// TIA Portal project "LabSupervision" (V16)

(* hardware
DEVICE "S71500/ET200MP station_1"  S7-1500 station
   slot 0: "Perfil soporte_0"  Rack  6ES7 590-1***0-0AA0
   slot 0: "PM 70W 120/230VAC"  PM 70W 120/230VAC  6EP1332-4BA00
   slot 1: "PLC_1"  CPU 1511-1 PN  6ES7 511-1AK00-0AB0  V1.0
      slot 3: "Display de la CPU_1"  6ES7591-1XA00-0AA0
      slot 32768: "Interfaz PROFINET_1"  X1
   slot 2: "CM 1542-5_1"  CM 1542-5  6GK7 542-5DX00-0XE0  V1.0
   slot 3: "DI 16x24VDC HF_1"  DI 16x24VDC HF  6ES7 521-1BH00-0AB0  V1.0
   slot 4: "DQ 16x24VDC/0.5A HF_1"  DQ 16x24VDC/0.5A HF  6ES7 522-1BH01-0AB0  V1.0
   slot 5: "AI 8xU/I/RTD/TC ST_1"  AI 8xU/I/RTD/TC ST  6ES7 531-7KF00-0AB0  V1.0
   slot 6: "AQ 4xU/I ST_1"  AQ 4xU/I ST  6ES7 532-5HD00-0AB0  V1.0
DEVICE "HMI_1"  KTP600 Basic color PN
   slot 0: "HMI_1"  KTP600 Basic color PN  6AV6 647-0AD11-3AX0  12.0.0.0
   slot 1: "HMI_RT_1"  KTP600 Basic color PN  6AV6 647-0AD11-3AX0  12.0.0.0
   slot 5: "HMI_1.IE_CP_1"  PROFINET Interface  12.0.0.0
      slot 1: "Interfaz PROFINET_1"  PROFINET Interface
         slot 1: "Port_1"  Port
DEVICE "PC-System_1"  SIMATIC PC station
   slot 0: "Estación PC SIMATIC"  Rail  SIMATIC PC-Station  V1.0
      slot 125: "Stationmanager"  Station_Manager  V6.0.4
   slot 1: "HMI_RT_2"  WinCC RT Professional  6AV2 105-0xxxx-xxxx  16.0.0.0
   slot 2: "IE general_1"  IE General  IE_CP  V8.2.0
DEVICE "SINAMICS G_1"  Sinamics.Device
   slot 0: "	_0"  Rail  SinamicsG120RackPN
   slot 0: "Accionamiento_1"  G120 CU240E-2 PN  6SL3244-0BB12-1FA0  4.7.6
      slot 1: "Interfaz PROFINET"  MDD-SinamicsG120-P
   slot 3: "PM240-2 IP20"  PM240-2 IP20  6SL3210-1PB13-8ULx  -
*)

// ===== PLC "PLC_1"  CPU 1511-1 PN =====

VAR_GLOBAL   // PLC tag table "Tabla de variables estándar"
   "Señal_Intermitente" AT %Q0.0 : Bool;
   "STAR" AT %M0.0 : Bool;
   "Potenciometro" AT %MW2 : Int;
   "Nivel_Actual" AT %QW2 : Int;
   "pot_Normalizado" AT %MD2 : Real;
   "Alarma_Nivel_Alto" AT %Q0.1 : Bool;
   "Alarma_Nivel_Bajo" AT %Q0.2 : Bool;
   "Stop" AT %I0.1 : Bool;
   "Paro_Emergencia" AT %I0.3 : Bool;
   "BomBa" AT %Q0.3 : Bool;
   "Sensor_Nivel_Alto" AT %I0.4 : Bool;
   "Sensor_Nivel_Bajo" AT %I0.5 : Bool;
   "Sistema" AT %M0.7 : Bool;
   "Bomba_Agua" AT %M0.2 : Bool;
   "Referencia" AT %MW6 : Int;
   "Nivel_Alcanzado" AT %Q0.6 : Bool;
   "Delante" AT %M0.6 : Bool;
   "Atras" AT %M1.0 : Bool;
   "RPM" AT %M8.0 : LReal;
END_VAR

DATA_BLOCK "Bloque_1_DB"   // DB5
{ S7_Optimized_Access := 'TRUE' }
VERSION : 0.1
// stored: InstanceOfName Bloque_1
"Bloque_1"
BEGIN
END_DATA_BLOCK

DATA_BLOCK "Base_Datos"   // DB8
{ S7_Optimized_Access := 'TRUE' }
VERSION : 0.1
   VAR
      RPM : Real;
      NivelLeidoInt : Real;
      Revoluciones_datos : Real;
   END_VAR
BEGIN
END_DATA_BLOCK

// folder: System blocks/Program resources

DATA_BLOCK "Encender"   // DB1
{ S7_Optimized_Access := 'TRUE' }
AUTHOR : Simatic
FAMILY : IEC
NAME : IEC_TMR
VERSION : 1.0
// stored: InstanceOfName IEC_TIMER
"IEC_TIMER"
BEGIN
END_DATA_BLOCK

DATA_BLOCK "apagar"   // DB2
{ S7_Optimized_Access := 'TRUE' }
AUTHOR : Simatic
FAMILY : IEC
NAME : IEC_TMR
VERSION : 1.0
// stored: InstanceOfName IEC_TIMER
"IEC_TIMER"
BEGIN
END_DATA_BLOCK

DATA_BLOCK "IEC_Timer_0_DB"   // DB3
{ S7_Optimized_Access := 'TRUE' }
AUTHOR : Simatic
FAMILY : IEC
NAME : IEC_TMR
VERSION : 1.0
// stored: InstanceOfName IEC_TIMER
"IEC_TIMER"
BEGIN
END_DATA_BLOCK

DATA_BLOCK "IEC_Timer_0_DB_1"   // DB6
{ S7_Optimized_Access := 'TRUE' }
AUTHOR : Simatic
FAMILY : IEC
NAME : IEC_TMR
VERSION : 1.0
// stored: InstanceOfName IEC_TIMER
"IEC_TIMER"
BEGIN
END_DATA_BLOCK

DATA_BLOCK "IEC_Timer_0_DB_2"   // DB7
{ S7_Optimized_Access := 'TRUE' }
AUTHOR : Simatic
FAMILY : IEC
NAME : IEC_TMR
VERSION : 1.0
// stored: InstanceOfName IEC_TIMER
"IEC_TIMER"
BEGIN
END_DATA_BLOCK

// folder: (top level)

DATA_BLOCK "TO_SpeedAxis_1"   // DB4, Motion_DB
{ S7_Optimized_Access := 'TRUE' }
AUTHOR : SIMATIC
FAMILY : MC_1500
VERSION : 1.0
// stored: InstanceOfName TO_SpeedAxis
"TO_SpeedAxis"
BEGIN
   DynamicLimits.MaxAcceleration := 1000.0;
   DynamicLimits.MaxDeceleration := 1000.0;
   DynamicLimits.MaxJerk := 20000.0;
   DynamicDefaults.Acceleration := 200.0;
   DynamicDefaults.Deceleration := 200.0;
   DynamicDefaults.Jerk := 4000.0;
   DynamicDefaults.EmergencyDeceleration := 1000.0;
   Actor.Interface.AddressOut := 256;
   Actor.Interface.AddressIn := 256;
END_DATA_BLOCK

FUNCTION_BLOCK "Bloque_1"   // FB1, LAD
{ S7_Optimized_Access := 'TRUE' }
VERSION : 0.1
   VAR
      MC_POWER_Instance : MC_POWER;
      MC_RESET_Instance : MC_RESET;
      MC_MOVEJOG_Instance : MC_MOVEJOG;
   END_VAR
BEGIN

REGION Network 1
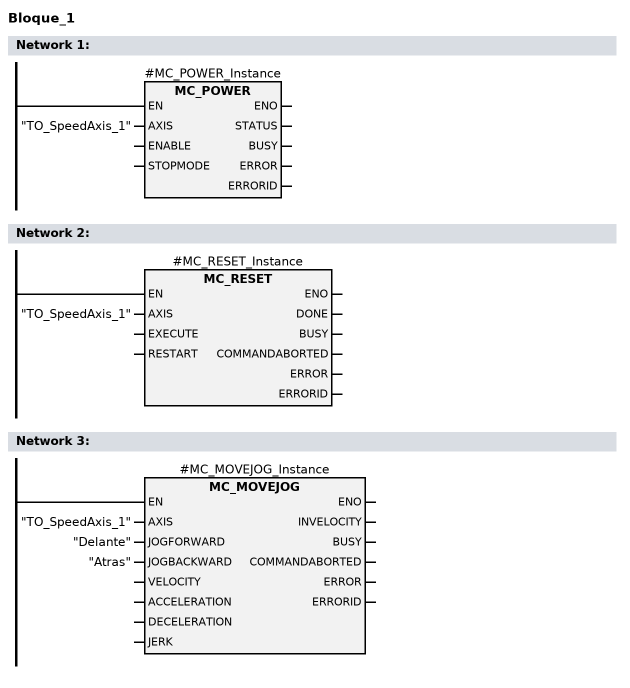
   #MC_POWER_Instance(Axis := "TO_SpeedAxis_1");   // MC_POWER
END_REGION

REGION Network 2
   #MC_RESET_Instance(Axis := "TO_SpeedAxis_1");   // MC_RESET
END_REGION

REGION Network 3
   #MC_MOVEJOG_Instance(Axis := "TO_SpeedAxis_1", JogForward := "Delante", JogBackward := "Atras");   // MC_MOVEJOG
END_REGION
END_FUNCTION_BLOCK

ORGANIZATION_BLOCK "Main"   // OB1, LAD, ProgramCycle
TITLE = "Main Program Sweep (Cycle)"
{ S7_Optimized_Access := 'TRUE' }
VERSION : 0.1
   VAR_INPUT
      Initial_Call : Bool;   // Initial call of this OB
      Remanence : Bool;   // =True, if remanent data are available
   END_VAR
   VAR_TEMP
      Temp_1 : Bool;
      Activar_Bomba : Bool;
      intermitencia : Bool;
   END_VAR
   VAR_TEMP   // added for the SCL form of the ladder/FBD networks
      _w1 : Bool;
   END_VAR
BEGIN

REGION Network 1: Normalizar Señal
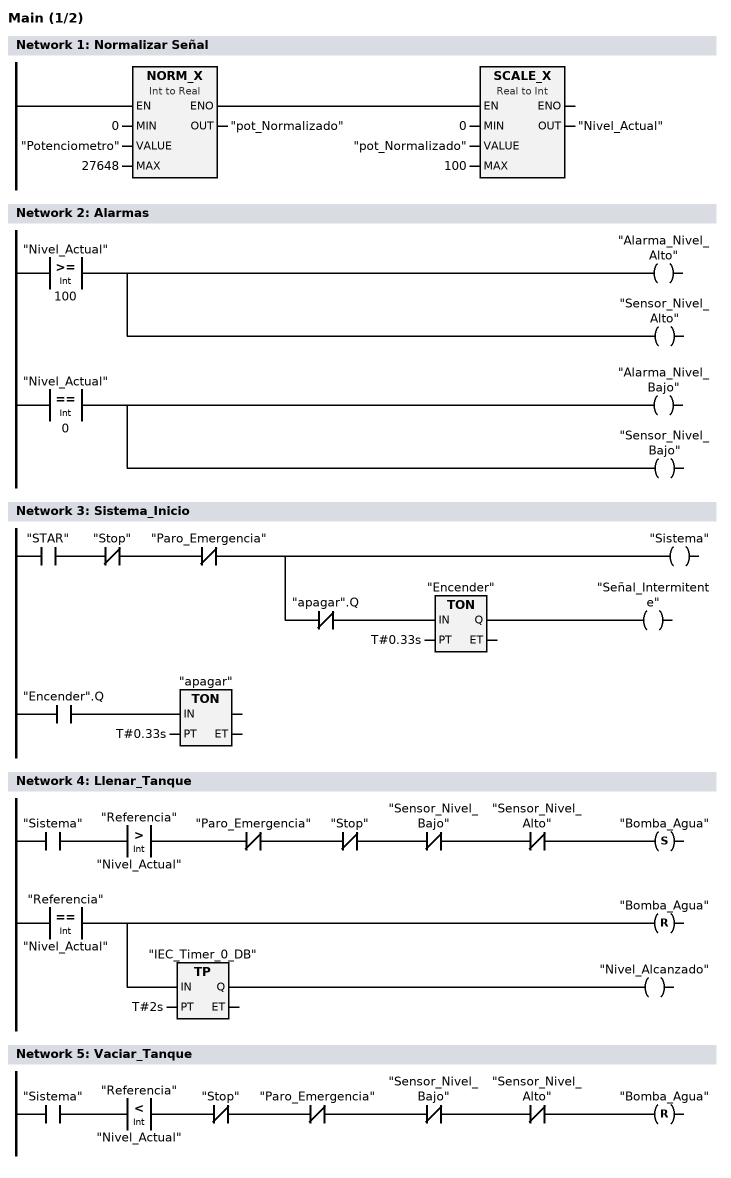
   RUNG wire#powerrail
      { S7_Templates := "[SrcType := Int, DestType := Real]" } Normalize(min := 0, value := "Potenciometro", max := 27648, out => "pot_Normalizado")
      { S7_Templates := "[SrcType := Real, DestType := Int]" } Scale(min := 0, value := "pot_Normalizado", max := 100, out => "Nivel_Actual")
   END_RUNG
   // the same network as SCL:
   "pot_Normalizado" := NORM_X(MIN := 0, VALUE := "Potenciometro", MAX := 27648);
   "Nivel_Actual" := SCALE_X(MIN := 0, VALUE := "pot_Normalizado", MAX := 100);
END_REGION

REGION Network 2: Alarmas
   RUNG wire#powerrail
      { S7_Templates := "SrcType := Int" } GE_Contact(in1 := "Nivel_Actual", in2 := 100)
      wire#w1
      Coil( "Alarma_Nivel_Alto" )
   END_RUNG
   RUNG wire#w1
      Coil( "Sensor_Nivel_Alto" )
   END_RUNG
   RUNG wire#powerrail
      { S7_Templates := "SrcType := Int" } EQ_Contact(in1 := "Nivel_Actual", in2 := 0)
      wire#w2
      Coil( "Alarma_Nivel_Bajo" )
   END_RUNG
   RUNG wire#w2
      Coil( "Sensor_Nivel_Bajo" )
   END_RUNG
   // the same network as SCL:
   "Alarma_Nivel_Alto" := "Nivel_Actual" >= 100;
   "Sensor_Nivel_Alto" := "Alarma_Nivel_Alto";
   "Alarma_Nivel_Bajo" := "Nivel_Actual" = 0;
   "Sensor_Nivel_Bajo" := "Alarma_Nivel_Bajo";
END_REGION

REGION Network 3: Sistema_Inicio
   "Sistema" := "STAR" AND NOT "Stop" AND NOT "Paro_Emergencia";
   "Encender".TON(IN := "Sistema" AND NOT "apagar".Q, PT := T#0.33s);
   "Señal_Intermitente" := "Encender".Q;
   "apagar".TON(IN := "Encender".Q, PT := T#0.33s);
END_REGION

REGION Network 4: Llenar_Tanque
   IF "Sistema" AND ("Referencia" > "Nivel_Actual") AND NOT "Paro_Emergencia" AND NOT "Stop" AND NOT "Sensor_Nivel_Bajo" AND NOT "Sensor_Nivel_Alto" THEN
       "Bomba_Agua" := TRUE;
   END_IF;
   #_w1 := "Referencia" = "Nivel_Actual";
   IF #_w1 THEN "Bomba_Agua" := FALSE; END_IF;
   "IEC_Timer_0_DB".TP(IN := #_w1, PT := T#2s);
   "Nivel_Alcanzado" := "IEC_Timer_0_DB".Q;
END_REGION

REGION Network 5: Vaciar_Tanque
   RUNG wire#powerrail
      Contact( "Sistema" )
      { S7_Templates := "SrcType := Int" } LT_Contact(in1 := "Referencia", in2 := "Nivel_Actual")
      I_Contact( "Stop" )
      I_Contact( "Paro_Emergencia" )
      I_Contact( "Sensor_Nivel_Bajo" )
      I_Contact( "Sensor_Nivel_Alto" )
      R_Coil( "Bomba_Agua" )
   END_RUNG
   // the same network as SCL:
   IF "Sistema" AND ("Referencia" < "Nivel_Actual") AND NOT "Stop" AND NOT "Paro_Emergencia" AND NOT "Sensor_Nivel_Bajo" AND NOT "Sensor_Nivel_Alto" THEN
       "Bomba_Agua" := FALSE;
   END_IF;
END_REGION

REGION Network 6: Variador
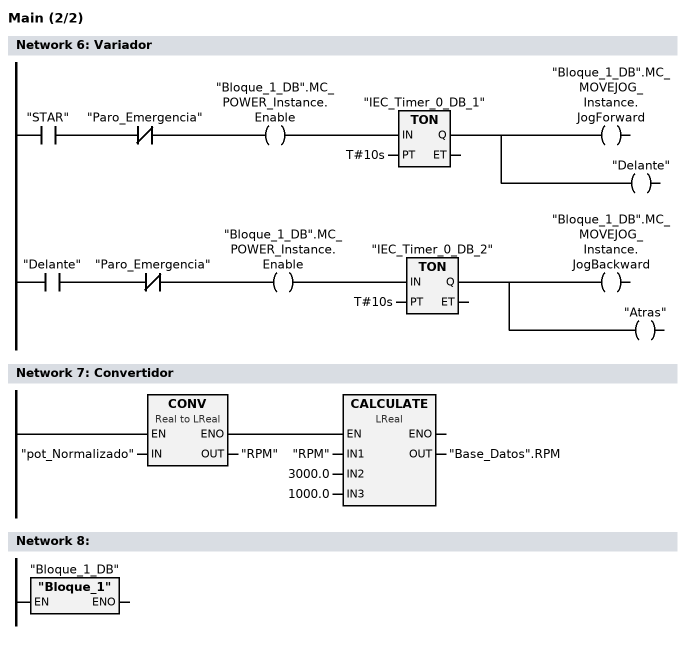
   "Bloque_1_DB".MC_POWER_Instance.Enable := "STAR" AND NOT "Paro_Emergencia";
   "IEC_Timer_0_DB_1".TON(IN := "Bloque_1_DB".MC_POWER_Instance.Enable, PT := T#10s);
   "Bloque_1_DB".MC_MOVEJOG_Instance.JogForward := "IEC_Timer_0_DB_1".Q;
   "Delante" := "IEC_Timer_0_DB_1".Q;
   "Bloque_1_DB".MC_POWER_Instance.Enable := "Delante" AND NOT "Paro_Emergencia";
   "IEC_Timer_0_DB_2".TON(IN := "Bloque_1_DB".MC_POWER_Instance.Enable, PT := T#10s);
   "Bloque_1_DB".MC_MOVEJOG_Instance.JogBackward := "IEC_Timer_0_DB_2".Q;
   "Atras" := "IEC_Timer_0_DB_2".Q;
END_REGION

REGION Network 7: Convertidor
   RUNG wire#powerrail
      { S7_Templates := "[SrcType := Real, DestType := LReal]" } Convert(in := "pot_Normalizado", out => "RPM")
      { S7_Templates := "SrcType := LReal"; S7_Expression := "(IN1+IN2)+(IN3)" } Calculate(in1 := "RPM", in2 := 3000.0, in3 := 1000.0, out => "Base_Datos".RPM)
   END_RUNG
   // the same network as SCL:
   "RPM" := REAL_TO_LREAL("pot_Normalizado");
   "Base_Datos".RPM := ("RPM"+3000.0)+(1000.0);
END_REGION

REGION Network 8
   RUNG wire#powerrail
      "Bloque_1_DB"()
   END_RUNG
   // the same network as SCL:
   "Bloque_1_DB"();   // "Bloque_1"
END_REGION
END_ORGANIZATION_BLOCK

(* ===== HMI "HMI_RT_1" =====
system functions are stored by id; their names below are inferred from use
connection "HMI_Conexión_1": ETHERNET, SMART_S7_1500_OMS

HMI tags "Tabla de variables estándar"
   "Número_imagen_variable" : UInt, internal
   "Nivel_Actual" : Int = PLC Nivel_Actual AT %QW2, 1 s
   "STAR" : Bool = PLC STAR AT %M0.0, 1 s
   "Stop" : Bool = PLC Stop AT %I0.1, 1 s
   "Bomba_Agua" : Bool = PLC Bomba_Agua AT %M0.2, 1 s
   "Sensor_Nivel_Bajo" : Bool = PLC Sensor_Nivel_Bajo AT %I0.5, 1 s
   "Sensor_Nivel_Alto" : Bool = PLC Sensor_Nivel_Alto AT %I0.4, 1 s
   "Paro_Emergencia" : Bool = PLC Paro_Emergencia AT %I0.3, 1 s
   "Referencia" : Int = PLC Referencia AT %MW6, 1 s
   "Señal_Intermitente" : Bool = PLC Señal_Intermitente AT %Q0.0, 1 s
   "Nivel_Alcanzado" : Bool = PLC Nivel_Alcanzado AT %Q0.6, 1 s
   "RPM" : LReal = PLC RPM AT %M8.0, 1 s

text list "Nombre_imagen_lista_texto": 1 'Imagen raíz'

Template "Plantilla_1" 320x240
   Button "Salir" at 266,202 size 52x37; TextOff 'Salir'; PictureOff "ExitRuntime_KTP600_Basic_color_PN"; PictureOn "ExitRuntime_KTP600_Basic_color_PN"
      on Release: StopRuntime(0)
   Button "Template_Button" at 213,202 size 52x37; TextOff 'Text'
   Button "Template_Button_1" at 160,202 size 52x37; TextOff 'Text'
   Button "Template_Button_2" at 107,202 size 52x37; TextOff 'Text'
   Button "Avisos" at 54,202 size 52x37; TextOff 'Avisos'; PictureOff "AlarmDisplay_KTP600_Basic_color_PN"; PictureOn "AlarmDisplay_KTP600_Basic_color_PN"
      on Release: function_ef3f5d25("Ventana de avisos_no_acusado", -1)
   Button "Imagen inicial" at 1,202 size 52x37; TextOff 'Imagen inicial'; PictureOff "NavigateHome_KTP600_Basic_color_PN"; PictureOn "NavigateHome_KTP600_Basic_color_PN"
      on Release: ActivateScreen("Control_Tanques", 0)
   SymbolicIOField "Imagen_campo_ES_simbólico" at 69,7 size 164x24; TextOff '0'; TextOn '1'; TextList "Nombre_imagen_lista_texto"
      ProcessValue <- "Número_imagen_variable"
      on Change: ActivateScreenByNumber("Número_imagen_variable", 0)
   DateTimeField "HmiScreenItemData" at 235,19 size 85x19
   DateTimeField "HmiScreenItemData_1" at 235,0 size 85x19
   GraphicView "Logotipo" at 0,0 size 67x38; Picture "Logotipo de HMI_1"

screen "Control_Tanques" 320x240, template "Plantilla_1"
   on GenerateScreen: SetTag("Número_imagen_variable", 1)
   Button "Botón_1" at 38,208 size 36x26; TextOff 'Star'
      on Press: SetBit("STAR")
   Button "Botón_2" at 84,209 size 32x25; TextOff 'Stop'
      on Press: InvertBit("Stop")
   Button "Botón_3" at 133,209 size 38x25; TextOff 'Paro'
      on Press: InvertBit("Paro_Emergencia")
   GraphicView "Visor de gráficos_6" at 70,58 size 91x84; Picture "Gráfico_29"
   GraphicView "Visor de gráficos_3" at 19,167 size 32x30; Picture "Gráfico_21"
      Visibility <- "Bomba_Agua"
   Bar "Barra_1" at 81,61 size 71x71; MinimumValue 0; MaximumValue 100
      ProcessValue <- "Nivel_Actual"
   GraphicView "Visor de gráficos_7" at 20,167 size 32x29; Picture "Gráfico_31"
      Visibility <- "Bomba_Agua"
   GraphicView "Visor de gráficos_8" at 67,160 size 19x24; Picture "Gráfico_27"
   GraphicView "Visor de gráficos_9" at 50,163 size 19x19; Picture "Gráfico_18"
   GraphicView "Visor de gráficos_1" at 3,168 size 17x19; Picture "Gráfico_18"
   GraphicView "Visor de gráficos_2" at 68,146 size 14x22; Picture "Gráfico_26"
   GraphicView "Visor de gráficos_11" at 190,59 size 30x27; Picture "Gráfico_34"
      Visibility <- "Sensor_Nivel_Alto"
   GraphicView "Visor de gráficos_4" at 16,131 size 34x30; Picture "Gráfico_34"
      Visibility <- "Sensor_Nivel_Bajo"
   GraphicView "Visor de gráficos_12" at 190,53 size 32x30; Picture "Gráfico_35"
      Visibility <- "Sensor_Nivel_Alto"
   GraphicView "Visor de gráficos_13" at 18,132 size 33x29; Picture "Gráfico_35"
      Visibility <- "Sensor_Nivel_Bajo"
   IOField "Campo ES_1" at 171,125 size 37x23; FormatPattern 999
      ProcessValue <- "Nivel_Actual"
   TrendView "Visor de curvas_1" at 212,87 size 103x89
   Circle "Círculo_2" at 181,7 size 27x27
      Appearance <- "Nivel_Alcanzado"
   TextField "Campo de texto_4" at 212,10 size 96x16; Text 'Nivel Alcanzado'
   Circle "Círculo_3" at 20,10 size 27x27
      Appearance <- "Señal_Intermitente"
   TextField "Campo de texto_5" at 58,17 size 39x16; Text 'Señal'
   Button "Botón_4" at 190,187 size 35x25; TextOff '+'
      on Click: function_dd21b452("Referencia", 1)
      on Press: function_dd21b452("Referencia", 1)
   Button "Botón_5" at 235,187 size 32x24; TextOff '-'
      on Click: function_b9b71300("Referencia", 1)
      on Press: function_b9b71300("Referencia", 1)
   IOField "Campo ES_2" at 273,185 size 37x23; FormatPattern 999
      ProcessValue <- "Referencia"
   IOField "Campo ES_3" at 171,152 size 37x23; FormatPattern 999
      ProcessValue <- "Referencia"
   IOField "Campo ES_4" at 265,37 size 37x23; FormatPattern 999999999.999
      ProcessValue <- "RPM"
   TextField "Campo de texto_1" at 220,33 size 30x16; Text 'RPM'
*)

(* ===== HMI "HMI_RT_2" =====
system functions are stored by id; their names below are inferred from use
connection "HMI_Conexión_2": S71200_TCP_IP, SCADA_S7_1500_OMS
connection "HMI_Conexión_3": S71200_TCP_IP, SCADA_S7_1500_OMS

HMI tags "Tabla de variables estándar"
   "Nivel_Actual" : Int = PLC Nivel_Actual AT %QW2, 500 ms
   "Referencia" : Int = PLC Referencia AT %MW6, 500 ms
   "Sensor_Nivel_Bajo" : Bool = PLC Sensor_Nivel_Bajo AT %I0.5, 500 ms
   "Sensor_Nivel_Alto" : Bool = PLC Sensor_Nivel_Alto AT %I0.4, 500 ms
   "Bomba_Agua" : Bool = PLC Bomba_Agua AT %M0.2, 500 ms
   "STAR" : Bool = PLC STAR AT %M0.0, 500 ms
   "Stop" : Bool = PLC Stop AT %I0.1, 500 ms
   "Paro_Emergencia" : Bool = PLC Paro_Emergencia AT %I0.3, 500 ms
   "Señal_Intermitente" : Bool = PLC Señal_Intermitente AT %Q0.0, 500 ms
   "Nivel_Alcanzado" : Bool = PLC Nivel_Alcanzado AT %Q0.6, 500 ms

screen "Control_Tanque" 1024x768
   Button "Botón_1" at 74,416 size 108x74; TextOff 'Star'
      on Press: SetBit("STAR")
      on Click: SetBit("STAR")
   Button "Botón_2" at 207,416 size 104x74; TextOff 'Stop'
      on Press: SetBit("Stop")
      on Click: InvertBit("Stop")
   Button "Botón_3" at 336,416 size 117x71; TextOff 'Paro'
      on Press: SetBit("Paro_Emergencia")
      on Click: InvertBit("Paro_Emergencia")
   TextField "Campo de texto_1" at 373,138 size 47x29; Text 'LEH'
   TextField "Campo de texto_2" at 58,172 size 43x29; Text 'LEL'
   GraphicView "Visor de gráficos_6" at 160,75 size 191x159; Picture "Gráfico_29"
   GraphicView "Visor de gráficos_3" at 64,293 size 81x92; Picture "Gráfico_21"
      Visibility <- "Bomba_Agua"
   Bar "Barra_1" at 186,90 size 125x132; MinimumValue 0; MaximumValue 100
      ProcessValue <- "Nivel_Actual"
   GraphicView "Visor de gráficos_7" at 48,295 size 97x91; Picture "Gráfico_31"
      Visibility <- "Bomba_Agua"
   TextField "Campo de texto_3" at 241,38 size 212x23; Text 'Sistema de Control Nivel'
   GraphicView "Visor de gráficos_8" at 178,280 size 78x54; Picture "Gráfico_27"
   GraphicView "Visor de gráficos_9" at 145,279 size 38x56; Picture "Gráfico_18"
   GraphicView "Visor de gráficos_2" at 182,226 size 69x61; Picture "Gráfico_26"
   GraphicView "Visor de gráficos_11" at 380,97 size 42x41; Picture "Gráfico_34"
      Visibility <- "Sensor_Nivel_Alto"
   GraphicView "Visor de gráficos_4" at 44,223 size 56x46; Picture "Gráfico_34"
      Visibility <- "Sensor_Nivel_Bajo"
   GraphicView "Visor de gráficos_12" at 380,94 size 49x44; Picture "Gráfico_35"
      Visibility <- "Sensor_Nivel_Alto"
   GraphicView "Visor de gráficos_13" at 43,222 size 56x47; Picture "Gráfico_35"
      Visibility <- "Sensor_Nivel_Bajo"
   IOField "Campo ES_1" at 513,355 size 75x48; FormatPattern 999
      ProcessValue <- "Referencia"
   WindowSlider "Barra de desplazamiento_1" at 523,220 size 47x124
      ProcessValue <- "Referencia"
   IOField "Campo ES_2" at 277,240 size 60x40; FormatPattern 999
      ProcessValue <- "Nivel_Actual"
   OnlineTrendControl "Visor de curvas f(t)_1" at 623,207 size 396x302
   Circle "Círculo_2" at 570,20 size 48x48
      Appearance <- "Nivel_Alcanzado"
   TextField "Campo de texto_4" at 541,85 size 120x18; Text 'Nivel Alcanzado'
   Circle "Círculo_1" at 738,17 size 48x48
      Appearance <- "Señal_Intermitente"
   TextField "Campo de texto_5" at 739,79 size 46x18; Text 'Señal'
   IOField "Campo ES_3" at 513,153 size 75x48; FormatPattern 999
      ProcessValue <- "Referencia"
   GraphicView "Visor de gráficos_1" at 1,293 size 51x56; Picture "Gráfico_18"
*)